{attribute addProperty BoxType "AMP8000-0030-0103-0103"}
{attribute addProperty Id "FSOEAT %I*FSOE_6FBCDF63162"}
{attribute addProperty CRC "171299057"}
{attribute addProperty SizeInBites "16"}
{attribute addProperty SizeInBytes "2"}
TYPE FSLOGIC_Inputs_0A35D0F1 :
STRUCT
	{attribute addProperty Name "FSOE"}
	FSOE AT %I* : FSOE_6FBCDF63;
END_STRUCT
END_TYPE

(* stored: Version 1.2.0.0, ProductVersion 3.1.4024.9
   DUT FSLOGIC_Inputs_0A35D0F1: Id {77ad4465-6b6c-4ba8-a7b6-830501ee2a1c} *)
